{attribute 'linkalways'} 
{attribute 'no_explicit_call' := 'This FB is a CLASS and must be accessed using methods or properties'}
{attribute 'enable_dynamic_creation'}
FUNCTION_BLOCK FINAL MOD_SINT EXTENDS Node
VAR
	in1 : _SINT(0);
	in2 : _SINT(0);
	out : _SINT(0);
END_VAR

METHOD PUBLIC Clone : I_Node
VAR
	pNode : POINTER TO MOD_SINT;
END_VAR
pNode := __NEW(MOD_SINT);
Clone := pNode^;
END_METHOD

METHOD FB_init : BOOL
VAR_INPUT
	bInitRetains : BOOL; // if TRUE, the retain variables are initialized (warm start / cold start)
	bInCopyCode : BOOL;  // if TRUE, the instance afterwards gets moved into the copy code (online change)
END_VAR
AddInput('in1',THIS^.in1);
AddInput('in2',THIS^.in2);
AddOutput('out', THIS^.out);
END_METHOD

METHOD PROTECTED OnExecute
VAR
END_VAR
out.Value := in1.Value MOD in2.Value;
END_METHOD

END_FUNCTION_BLOCK

(* stored: Version 1.1.0.1, ProductVersion 3.1.4024.15
   POU MOD_SINT: Id {960d3021-62dd-4c32-bcc1-eef723803c38}, SpecialFunc None
   Folder Constructor: Id {07a11c76-7852-4fba-ab45-cca43b6fa1fd}
   Method Clone: Id {e8cc7253-8892-47a1-8e85-4330d37e72eb}
   Method FB_init: Id {51360f92-ee1c-4788-ab0f-8171abb1d4a1}
   Method OnExecute: Id {108694d9-e9fd-4d91-8166-1bedb4bcdf72} *)
